Staubli VAL3: iGripOpen.pgx

public program iGripOpen(num& nNum[] (dimensions=1))
begin
  nNum=dioGet(iGripOpen)
end
